% RSLogix 500 project I2P-JOB-13 PART 2 DUNCAN_SUTTON.RSS, saved by version 10.00.00.00 %
PROJECT "ML01A"    % processor: Bul.1763 MicroLogix 1100 Series B %

PROGRAM FILES
  LAD 2   13 rungs

DATA FILES
  O0 OUTPUT  4 elements
  I1 INPUT  6 elements
  S2 STATUS  66 elements
  B3 BINARY  1 elements
  T4 TIMER  1 elements
  C5 COUNTER  1 elements
  R6 CONTROL  1 elements
  N7 INTEGER  1 elements
  F8 FLOAT  1 elements

LADDER 2
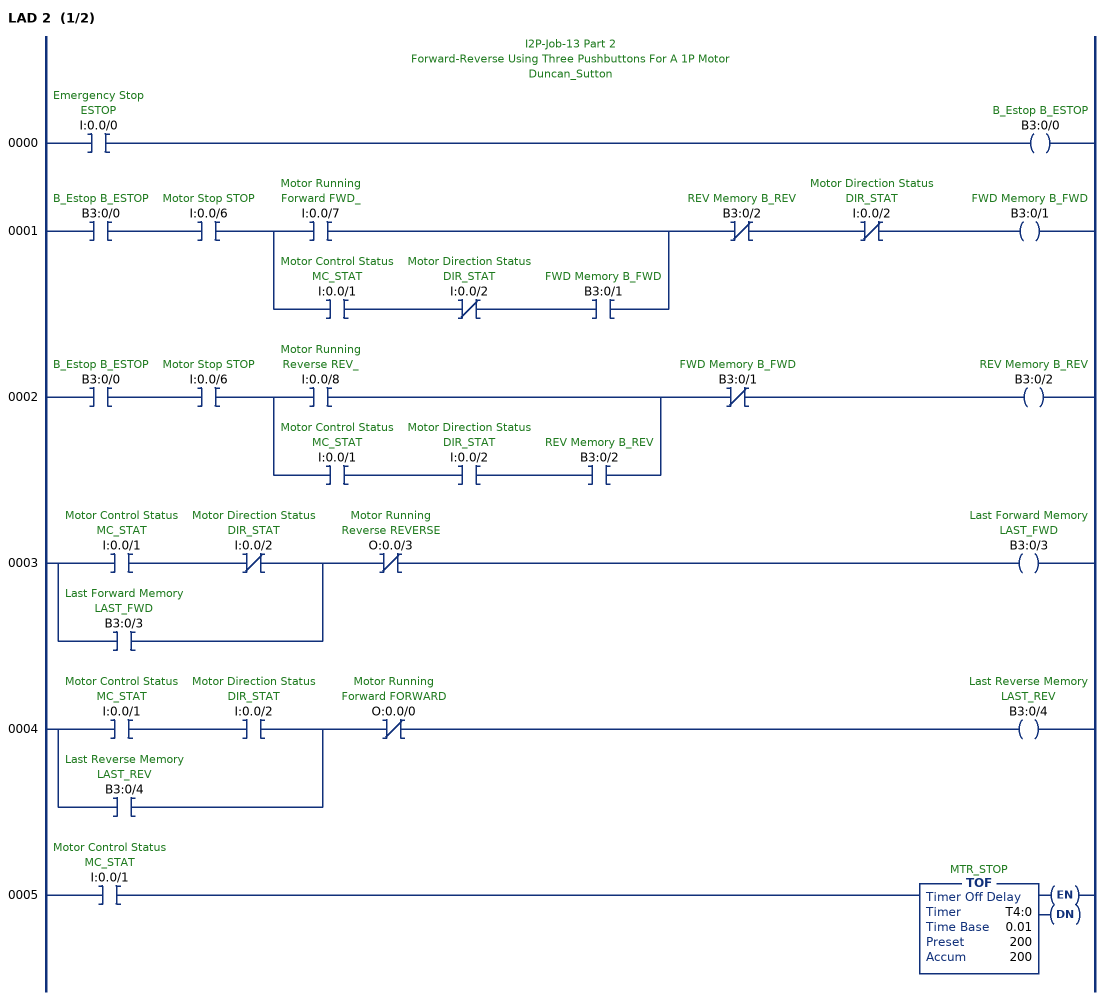
% Rung: 0 %
% I2P-Job-13 Part 2
% Forward-Reverse Using Three Pushbuttons For A 1P Motor
% Duncan_Sutton %
SOR XIC I:0.0/0 OTE B3:0/0 EOR
%   I:0.0/0  ESTOP  "Emergency Stop" %
%   B3:0/0  B_ESTOP  "B_Estop" %
% Rung: 1 %
SOR XIC B3:0/0 XIC I:0.0/6 BST XIC I:0.0/7 NXB XIC I:0.0/1 XIO I:0.0/2 XIC B3:0/1 BND XIO B3:0/2 XIO I:0.0/2 OTE B3:0/1 EOR
%   B3:0/0  B_ESTOP  "B_Estop" %
%   I:0.0/6  STOP  "Motor Stop" %
%   I:0.0/7  FWD_  "Motor Running Forward" %
%   I:0.0/1  MC_STAT  "Motor Control Status" %
%   I:0.0/2  DIR_STAT  "Motor Direction Status" %
%   B3:0/1  B_FWD  "FWD Memory" %
%   B3:0/2  B_REV  "REV Memory" %
% Rung: 2 %
SOR XIC B3:0/0 XIC I:0.0/6 BST XIC I:0.0/8 NXB XIC I:0.0/1 XIC I:0.0/2 XIC B3:0/2 BND XIO B3:0/1 OTE B3:0/2 EOR
%   B3:0/0  B_ESTOP  "B_Estop" %
%   I:0.0/6  STOP  "Motor Stop" %
%   I:0.0/8  REV_  "Motor Running Reverse" %
%   I:0.0/1  MC_STAT  "Motor Control Status" %
%   I:0.0/2  DIR_STAT  "Motor Direction Status" %
%   B3:0/2  B_REV  "REV Memory" %
%   B3:0/1  B_FWD  "FWD Memory" %
% Rung: 3 %
SOR BST XIC I:0.0/1 XIO I:0.0/2 NXB XIC B3:0/3 BND XIO O:0.0/3 OTE B3:0/3 EOR
%   I:0.0/1  MC_STAT  "Motor Control Status" %
%   I:0.0/2  DIR_STAT  "Motor Direction Status" %
%   B3:0/3  LAST_FWD  "Last Forward Memory" %
%   O:0.0/3  REVERSE  "Motor Running Reverse" %
% Rung: 4 %
SOR BST XIC I:0.0/1 XIC I:0.0/2 NXB XIC B3:0/4 BND XIO O:0.0/0 OTE B3:0/4 EOR
%   I:0.0/1  MC_STAT  "Motor Control Status" %
%   I:0.0/2  DIR_STAT  "Motor Direction Status" %
%   B3:0/4  LAST_REV  "Last Reverse Memory" %
%   O:0.0/0  FORWARD  "Motor Running Forward" %
% Rung: 5 %
SOR XIC I:0.0/1 TOF T4:0 0.01 200 200 EOR
%   I:0.0/1  MC_STAT  "Motor Control Status" %
%   T4:0  MTR_STOP %

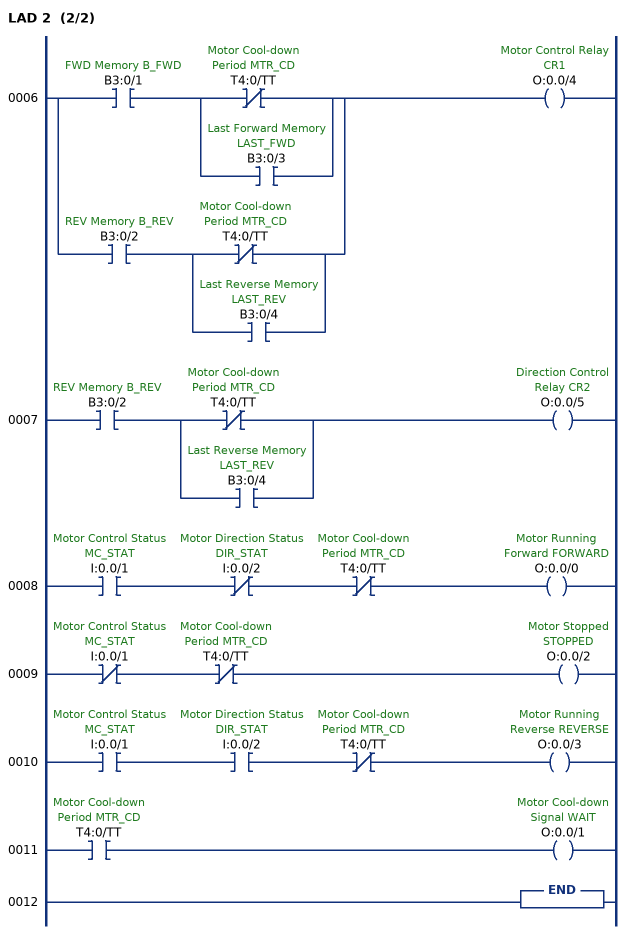
% Rung: 6 %
SOR BST XIC B3:0/1 BST XIO T4:0/TT NXB XIC B3:0/3 BND NXB XIC B3:0/2 BST XIO T4:0/TT NXB XIC B3:0/4 BND BND OTE O:0.0/4 EOR
%   B3:0/1  B_FWD  "FWD Memory" %
%   T4:0/TT  MTR_CD  "Motor Cool-down Period" %
%   B3:0/3  LAST_FWD  "Last Forward Memory" %
%   B3:0/2  B_REV  "REV Memory" %
%   B3:0/4  LAST_REV  "Last Reverse Memory" %
%   O:0.0/4  CR1  "Motor Control Relay" %
% Rung: 7 %
SOR XIC B3:0/2 BST XIO T4:0/TT NXB XIC B3:0/4 BND OTE O:0.0/5 EOR
%   B3:0/2  B_REV  "REV Memory" %
%   T4:0/TT  MTR_CD  "Motor Cool-down Period" %
%   B3:0/4  LAST_REV  "Last Reverse Memory" %
%   O:0.0/5  CR2  "Direction Control Relay" %
% Rung: 8 %
SOR XIC I:0.0/1 XIO I:0.0/2 XIO T4:0/TT OTE O:0.0/0 EOR
%   I:0.0/1  MC_STAT  "Motor Control Status" %
%   I:0.0/2  DIR_STAT  "Motor Direction Status" %
%   T4:0/TT  MTR_CD  "Motor Cool-down Period" %
%   O:0.0/0  FORWARD  "Motor Running Forward" %
% Rung: 9 %
SOR XIO I:0.0/1 XIO T4:0/TT OTE O:0.0/2 EOR
%   I:0.0/1  MC_STAT  "Motor Control Status" %
%   T4:0/TT  MTR_CD  "Motor Cool-down Period" %
%   O:0.0/2  STOPPED  "Motor Stopped" %
% Rung: 10 %
SOR XIC I:0.0/1 XIC I:0.0/2 XIO T4:0/TT OTE O:0.0/3 EOR
%   I:0.0/1  MC_STAT  "Motor Control Status" %
%   I:0.0/2  DIR_STAT  "Motor Direction Status" %
%   T4:0/TT  MTR_CD  "Motor Cool-down Period" %
%   O:0.0/3  REVERSE  "Motor Running Reverse" %
% Rung: 11 %
SOR XIC T4:0/TT OTE O:0.0/1 EOR
%   T4:0/TT  MTR_CD  "Motor Cool-down Period" %
%   O:0.0/1  WAIT  "Motor Cool-down Signal" %
% Rung: 12 %
SOR END EOR

OTHER DOCUMENTED ADDRESSES
  I:0.0/3  FWD  "Direction"
  I:0.0/4  REV  "Direction"
  I:0.0/5  2PSS_PA  "2 Poistion Selector Switch Position A"
  TT  "TOF/1 Timer"

DATA TABLE (non-zero values as saved)
DATA B3
% B3:0 % 0X0011
DATA T4
% .PRE .ACC %
% T4:0 % 200 200
